	16#4B75: sMsg := '4B75 parameter ST_NciTangentialFollowingDesc: nPathAxis1 and nPathAxis2, resp. are no path axes. So it is not possible to determine the plane.';
	16#4B76: sMsg := '4B76 parameter ST_NciTangentialFollwoingDesc: nPathAxis1 and nPathAxis2 are equal. So it is not possible to determine the plane.';
	16#4B77: sMsg := '4B77 parameter ST_NciGeoCirclePlane: circle is programmed in a wrong manner.';
	16#4B78: sMsg := '4B78 function Internal error in calculation of the tangential following';
	16#4B79: sMsg := '4B79 monitoring Tangential following: With ST_NciTangentialFollowingDesc the monitoring of the deviation angle (E_TfErrorOnCrirical1) is activated and with the actual segment the deviation angle is too big.';
	16#4B7A: sMsg := '4B7A function not implemented';
	16#4B7B: sMsg := '4B7B parameter Tangential Following: The radius of the actual circle segment is too small';
	16#4B7C: sMsg := '4B7C parameter FB_NciFeedTablePreparation: pEntry is NULL';
	16#4B7D: sMsg := '4B7D parameter FB_NciFeedTablePreparation: The specified nEntryType does not match the the structure type';
	16#4B7E: sMsg := '4B7E parameter ST_NciMFuncFast and ST_NciMFuncHsk: The requested m-function is not in between 0..159';
	16#4B7F: sMsg := '4B7F parameter ST_NciDynOvr: The requested value for the dynamic override is not in between 0.01 and 1.0';
	16#4B80: sMsg := '4B80 parameter ST_NciVertexSmoothing: invalid parameter. This error occurs with a negative vertex radius or an unknown vertex smoothing type.';
	16#4B81: sMsg := '4B81 parameter FB_NciFeedTablePrepartion: The requested velocity is not in a valid range';
	16#4B82: sMsg := '4B82 parameter ST_Nci*: invalid parameter';

ELSE
	sMsg := UDINT_TO_STRING(iErrID);
	sMsg := concat(sMsg, ' Unknown Error code');
END_CASE
F_AxErrMsg := sMsg;

END_FUNCTION

(* stored: Version 1.1.0.1, ProductVersion 3.1.4026.13, FileIdentifier 141133da2f31b8bb0962f54e5300aa364176dbc4, FileSignature 2a1a89e3e0b37524b411073874873a7b1e5f265d6b539e4a6338a2b25cc3e9fdc02ae217577785b81855868b4615aa780d4c27f8efc194135ffdfbb13e3ab8f6a5d5299821e3426d9f989205bca6eb758ebbac3b1f315423eda7f9755f7c60c9653cbe3c00a903d6d701e9259e6379704a170e82c78dc422f20dceaafa3c94a569448724ed37bc8dc9bf97e4323fb460199f7a6b571e9c0c029bccec6516802f0131f881df868ac86fbd66ec96d9c6c169140086fa27f9d3310666c5853ef738b55d76cb9890bbac9bd55a8305ee5a9249e4794c9dfd677a82d8881055cd5a2d33cd9eb2a17c5a96f7d53afbe5137f677967361e34032baf9c134793b2b1c5f5
   POU F_AxErrMsg: Id {06508107-56b8-4212-aec4-06150cd92788}, SpecialFunc None *)
